// 40 Visualizations/CLIENT/SERIAL Client/SERIAL Client/POPUP/PARAMETER/VIS_ModBusParameter_SERIAL_Client
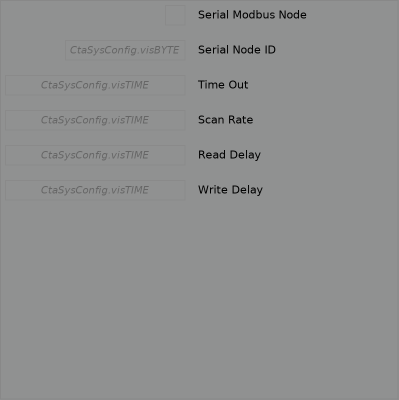
VISUALIZATION VIS_ModBusParameter_SERIAL_Client  // 399x400
VAR_IN_OUT
    fbMbSerialClientIn   : fbMbSerialClient; 
END_VAR
    Label (195,5 195x20), "Serial Modbus Node"
    Label (195,40 195x20), "Serial Node ID"
    Frame (65,40 120x20)
        shows CtaSysConfig.visBYTE(visfbBYTEIn := fbMbSerialClientIn.scParameter.fbbyUnitId)
    Frame (165,5 20x20)
        shows CtaSysConfig.visBOOL(visfbBOOLIn := fbMbSerialClientIn.scParameter.fbxEnable)
    Label (195,75 195x20), "Time Out"
    Frame (5,75 180x20)
        shows CtaSysConfig.visTIME(visfbTIMEIn := fbMbSerialClientIn.scParameter.fbtTimeOut)
    Frame (5,110 180x20)
        shows CtaSysConfig.visTIME(visfbTIMEIn := fbMbSerialClientIn.scParameter.fbtScanRate)
    Label (195,110 195x20), "Scan Rate"
    Frame (5,145 180x20)
        shows CtaSysConfig.visTIME(visfbTIMEIn := fbMbSerialClientIn.scParameter.fbtDelayRead)
    Label (195,145 195x20), "Read Delay"
    Frame (5,180 180x20)
        shows CtaSysConfig.visTIME(visfbTIMEIn := fbMbSerialClientIn.scParameter.fbtDelayWrite)
    Label (195,180 195x20), "Write Delay"
END_VISUALIZATION

// 40 Visualizations/CLIENT/NETWORK Client/TCP/VIS_ModBusTcpNode_QUERRY
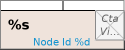
VISUALIZATION VIS_ModBusTcpNode_QUERRY  // 125x50
VAR_IN_OUT
	fbMbTcpClientIn   : REFERENCE TO fbMbTcpClient;      
END_VAR
    RoundedRectangle (0,10 125x40), colour toggle: fbMbTcpClientIn.xError
    RoundedRectangle (0,10 125x40), colour toggle: fbMbTcpClientIn.xError, invisible if: fbMbTcpClientIn.xComAktive
    Image (95,10 30x30), image: CtaVisSymbols.ImagePool.gear
        OnMouseClick:  Dialog=VIS_ModBus_Tcpl_NodePopUp, Parameters={fbMbTcpClientIn: fbMbTcpClientIn}, Selected={0: }, OpenModal=True, OpenCentered=True
    Textfield (30,37 90x10), "Node Id %d", text variable: fbMbTcpClientIn.byUnitId, invisible if: NOT __ISVALIDREF(fbMbTcpClientIn)
    Line (63,10) (63,0)
    Frame (5,15 80x20)
        shows Node_BMK(ITF_BMK := fbMbTcpClientIn.proITF_BMK)
END_VISUALIZATION

// 40 Visualizations/CLIENT/NETWORK Client/TCP/VIS_ModBusTcpNode
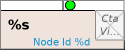
VISUALIZATION VIS_ModBusTcpNode  // 125x50
VAR_INPUT   
	ITF_TCP_NODEIN :   ITF_TCP_NODE;   
    xCourrentNode     :   BOOL;
END_VAR
    Frame (0,0 125x50), invisible if: NOT __QUERYINTERFACE(ITF_TCP_NODEIN,ITF_TCP_NODEIN)
        shows VIS_ModBusTcpNode_QUERRY(fbMbTcpClientIn := ITF_TCP_NODEIN.proNodeReference)
    Ellipse (65,0 10x10), invisible if: NOT xCourrentNode
END_VISUALIZATION

// 40 Visualizations/CLIENT/NETWORK Client/TCP/POPUP/VIS_ModBus_Tcpl_NodePopUp
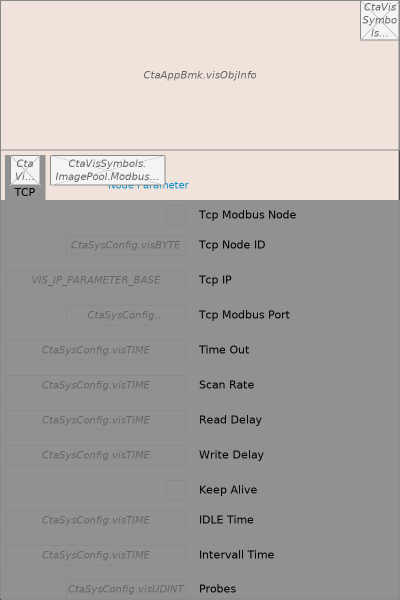
VISUALIZATION VIS_ModBus_Tcpl_NodePopUp  // 400x600
VAR_IN_OUT
    {attribute 'VAR_IN_OUT_AS_POINTER'}
	fbMbTcpClientIn   : fbMbTcpClient; 
END_VAR
    Rectangle (0,0 400x600)
    Label (105,180 150x10), "Node Parameter"
    Image (50,155 115x30), image: CtaVisSymbols.ImagePool.Modbus_Organization_Logo
    Group (5,155 40x45)
        Rectangle (0,0 40x45)
        Label (5,30 30x15), "TCP"
        Image (5,0 30x30), image: CtaVisSymbols.ImagePool.lan
    Frame (1,200 399x400)
        shows VIS_ModBusParameter_TCP_Client(fbMbTcpClientIn := fbMbTcpClientIn)
        shows VIS_ModBusParameter_UDP(fbModBusServerIn := fbModBusServerIn)
        shows VIS_ModBusParameter_SERIAL(fbModBusServerIn := fbModBusServerIn)
    Image (360,0 40x40), image: CtaVisSymbols.ImagePool.close_solo_black
        OnMouseClick:  Dialog=VIS_ModBus_Tcpl_NodePopUp, Result=None, NumpadKeypadSet=True
    Frame (0,0 400x150)
        shows CtaAppBmk.visObjInfo(ITF_BMK_IN := fbMbTcpClientIn.proITF_BMK)
END_VISUALIZATION

// 40 Visualizations/CLIENT/NETWORK Client/TCP/POPUP/PARAMETER/VIS_ModBusParameter_TCP_Client
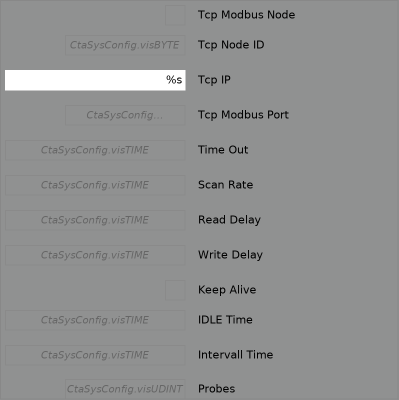
VISUALIZATION VIS_ModBusParameter_TCP_Client  // 399x400
VAR_IN_OUT
    fbMbTcpClientIn   : fbMbTcpClient; 
END_VAR
    Label (195,5 195x20), "Tcp Modbus Node"
    Label (195,35 195x20), "Tcp Node ID"
    Frame (65,35 120x20)
        shows CtaSysConfig.visBYTE(visfbBYTEIn := fbMbTcpClientIn.scParameter.fbbyUnitId)
    Frame (165,5 20x20)
        shows CtaSysConfig.visBOOL(visfbBOOLIn := fbMbTcpClientIn.scParameter.fbxEnable)
    Label (195,140 195x20), "Time Out"
    Frame (5,140 180x20)
        shows CtaSysConfig.visTIME(visfbTIMEIn := fbMbTcpClientIn.scParameter.fbtTimeOut)
    Frame (5,175 180x20)
        shows CtaSysConfig.visTIME(visfbTIMEIn := fbMbTcpClientIn.scParameter.fbtScanRate)
    Label (195,175 195x20), "Scan Rate"
    Frame (5,70 180x20)
        shows VIS_IP_PARAMETER(ITF_STRING40In := fbMbTcpClientIn.scParameter.fbstIp)
    Label (195,70 195x20), "Tcp IP"
    Frame (65,105 120x20)
        shows CtaSysConfig.visWORD_DEZ(visfbWORDIn := fbMbTcpClientIn.scParameter.fbwPort)
    Label (195,105 195x20), "Tcp Modbus Port"
    Frame (165,280 20x20)
        shows CtaSysConfig.visBOOL(visfbBOOLIn := fbMbTcpClientIn.scParameter.fbxKeepAlive)
    Label (195,280 195x20), "Keep Alive"
    Frame (5,310 180x20)
        shows CtaSysConfig.visTIME(visfbTIMEIn := fbMbTcpClientIn.scParameter.fbtMaxIdleTime)
    Label (195,310 195x20), "IDLE Time"
    Label (195,345 195x20), "Intervall Time"
    Frame (5,345 180x20)
        shows CtaSysConfig.visTIME(visfbTIMEIn := fbMbTcpClientIn.scParameter.fbtIntervall)
    Frame (65,379 120x20)
        shows CtaSysConfig.visUDINT(visfbUDINTIn := fbMbTcpClientIn.scParameter.fbudiProbes)
    Label (195,379 195x20), "Probes"
    Frame (5,210 180x20)
        shows CtaSysConfig.visTIME(visfbTIMEIn := fbMbTcpClientIn.scParameter.fbtDelayRead)
    Label (195,210 195x20), "Read Delay"
    Frame (5,245 180x20)
        shows CtaSysConfig.visTIME(visfbTIMEIn := fbMbTcpClientIn.scParameter.fbtDelayWrite)
    Label (195,245 195x20), "Write Delay"
END_VISUALIZATION

// 40 Visualizations/CLIENT/NETWORK Client/VIS_MODBUS_TCP_LINE
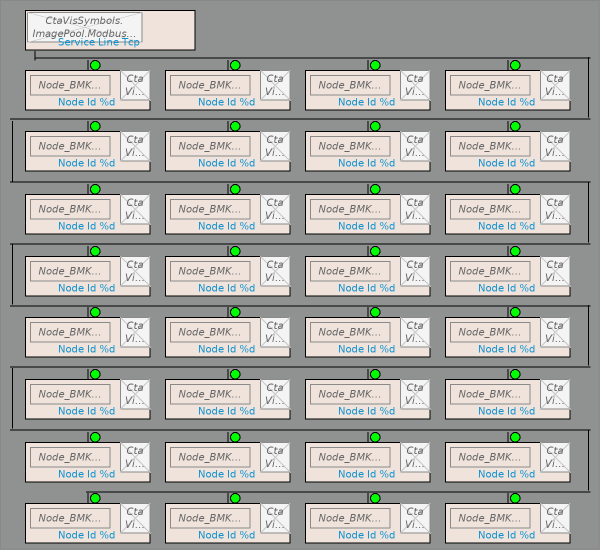
VISUALIZATION VIS_MODBUS_TCP_LINE  // 600x550
VAR_IN_OUT
	fbMbTcpPortControll   : fbMbTcpPortControll;      
END_VAR
    Frame (509,56 81x4), invisible if: fbMbTcpPortControll.bCountetCalls < 5
        shows VIS_TCP_LINE_HORIZONTAL()
    Frame (369,56 141x4), invisible if: fbMbTcpPortControll.bCountetCalls < 4
        shows VIS_TCP_LINE_HORIZONTAL()
    Frame (25,10 170x50)
        shows VIS_ModBusNetworkPortTcp(fbMbTcpPortControllIn := fbMbTcpPortControll)
    Frame (194,56 36x4), invisible if: fbMbTcpPortControll.bCountetCalls < 2
        shows VIS_TCP_LINE_HORIZONTAL()
    Frame (586,57 4x60), invisible if: fbMbTcpPortControll.bCountetCalls < 5
        shows VIS_TCP_LINE_VERTIKAL()
    Frame (10,121 4x60), invisible if: fbMbTcpPortControll.bCountetCalls < 9
        shows VIS_TCP_LINE_VERTIKAL()
    Frame (10,180 80x4), invisible if: fbMbTcpPortControll.bCountetCalls < 9
        shows VIS_TCP_LINE_HORIZONTAL()
    Frame (586,182 4x60), invisible if: fbMbTcpPortControll.bCountetCalls < 13
        shows VIS_TCP_LINE_VERTIKAL()
    Frame (10,244 4x60), invisible if: fbMbTcpPortControll.bCountetCalls < 17
        shows VIS_TCP_LINE_VERTIKAL()
    Frame (586,305 4x60), invisible if: fbMbTcpPortControll.bCountetCalls < 21
        shows VIS_TCP_LINE_VERTIKAL()
    Frame (10,368 4x60), invisible if: fbMbTcpPortControll.bCountetCalls < 25
        shows VIS_TCP_LINE_VERTIKAL()
    Frame (586,430 4x60), invisible if: fbMbTcpPortControll.bCountetCalls < 29
        shows VIS_TCP_LINE_VERTIKAL()
    Frame (229,56 141x4), invisible if: fbMbTcpPortControll.bCountetCalls < 3
        shows VIS_TCP_LINE_HORIZONTAL()
    Frame (506,117 84x4), invisible if: fbMbTcpPortControll.bCountetCalls < 5
        shows VIS_TCP_LINE_HORIZONTAL()
    Frame (366,117 141x4), invisible if: fbMbTcpPortControll.bCountetCalls < 6
        shows VIS_TCP_LINE_HORIZONTAL()
    Frame (86,117 141x4), invisible if: fbMbTcpPortControll.bCountetCalls < 8
        shows VIS_TCP_LINE_HORIZONTAL()
    Frame (226,117 141x4), invisible if: fbMbTcpPortControll.bCountetCalls < 7
        shows VIS_TCP_LINE_HORIZONTAL()
    Frame (10,117 77x4), invisible if: fbMbTcpPortControll.bCountetCalls < 9
        shows VIS_TCP_LINE_HORIZONTAL()
    Frame (89,180 141x4), invisible if: fbMbTcpPortControll.bCountetCalls < 10
        shows VIS_TCP_LINE_HORIZONTAL()
    Frame (229,180 141x4), invisible if: fbMbTcpPortControll.bCountetCalls < 11
        shows VIS_TCP_LINE_HORIZONTAL()
    Frame (509,180 81x4), invisible if: fbMbTcpPortControll.bCountetCalls < 13
        shows VIS_TCP_LINE_HORIZONTAL()
    Frame (369,180 141x4), invisible if: fbMbTcpPortControll.bCountetCalls < 12
        shows VIS_TCP_LINE_HORIZONTAL()
    Frame (506,242 84x4), invisible if: fbMbTcpPortControll.bCountetCalls < 13
        shows VIS_TCP_LINE_HORIZONTAL()
    Frame (366,242 141x4), invisible if: fbMbTcpPortControll.bCountetCalls < 14
        shows VIS_TCP_LINE_HORIZONTAL()
    Frame (86,242 141x4), invisible if: fbMbTcpPortControll.bCountetCalls < 16
        shows VIS_TCP_LINE_HORIZONTAL()
    Frame (226,242 141x4), invisible if: fbMbTcpPortControll.bCountetCalls < 15
        shows VIS_TCP_LINE_HORIZONTAL()
    Frame (10,242 77x4), invisible if: fbMbTcpPortControll.bCountetCalls < 17
        shows VIS_TCP_LINE_HORIZONTAL()
    Frame (10,304 80x4), invisible if: fbMbTcpPortControll.bCountetCalls < 17
        shows VIS_TCP_LINE_HORIZONTAL()
    Frame (89,304 141x4), invisible if: fbMbTcpPortControll.bCountetCalls < 18
        shows VIS_TCP_LINE_HORIZONTAL()
    Frame (229,304 141x4), invisible if: fbMbTcpPortControll.bCountetCalls < 19
        shows VIS_TCP_LINE_HORIZONTAL()
    Frame (509,304 81x4), invisible if: fbMbTcpPortControll.bCountetCalls < 21
        shows VIS_TCP_LINE_HORIZONTAL()
    Frame (369,304 141x4), invisible if: fbMbTcpPortControll.bCountetCalls < 20
        shows VIS_TCP_LINE_HORIZONTAL()
    Frame (506,365 84x4), invisible if: fbMbTcpPortControll.bCountetCalls < 21
        shows VIS_TCP_LINE_HORIZONTAL()
    Frame (366,365 141x4), invisible if: fbMbTcpPortControll.bCountetCalls < 22
        shows VIS_TCP_LINE_HORIZONTAL()
    Frame (86,365 141x4), invisible if: fbMbTcpPortControll.bCountetCalls < 24
        shows VIS_TCP_LINE_HORIZONTAL()
    Frame (226,365 141x4), invisible if: fbMbTcpPortControll.bCountetCalls < 23
        shows VIS_TCP_LINE_HORIZONTAL()
    Frame (10,365 77x4), invisible if: fbMbTcpPortControll.bCountetCalls < 25
        shows VIS_TCP_LINE_HORIZONTAL()
    Frame (10,428 80x4), invisible if: fbMbTcpPortControll.bCountetCalls < 25
        shows VIS_TCP_LINE_HORIZONTAL()
    Frame (89,428 141x4), invisible if: fbMbTcpPortControll.bCountetCalls < 26
        shows VIS_TCP_LINE_HORIZONTAL()
    Frame (229,428 141x4), invisible if: fbMbTcpPortControll.bCountetCalls < 27
        shows VIS_TCP_LINE_HORIZONTAL()
    Frame (509,428 81x4), invisible if: fbMbTcpPortControll.bCountetCalls < 29
        shows VIS_TCP_LINE_HORIZONTAL()
    Frame (369,428 141x4), invisible if: fbMbTcpPortControll.bCountetCalls < 28
        shows VIS_TCP_LINE_HORIZONTAL()
    Frame (506,490 84x4), invisible if: fbMbTcpPortControll.bCountetCalls < 29
        shows VIS_TCP_LINE_HORIZONTAL()
    Frame (366,490 141x4), invisible if: fbMbTcpPortControll.bCountetCalls < 30
        shows VIS_TCP_LINE_HORIZONTAL()
    Frame (86,490 141x4), invisible if: fbMbTcpPortControll.bCountetCalls < 32
        shows VIS_TCP_LINE_HORIZONTAL()
    Frame (226,490 141x4), invisible if: fbMbTcpPortControll.bCountetCalls < 31
        shows VIS_TCP_LINE_HORIZONTAL()
    Frame (25,60 125x50), invisible if: NOT fbMbTcpPortControll.ayShowNodes[1]
        shows VIS_ModBusTcpNode(ITF_TCP_NODEIN := fbMbTcpPortControll.ayNodes[1], xCourrentNode := fbMbTcpPortControll.bIdOfCourrentCall = 1)
        shows VIS_ModBusTcpNode()
        p1371288417: fbMbSerialPortControllIn.ayNodes[1]
    Frame (305,60 125x50), invisible if: NOT fbMbTcpPortControll.ayShowNodes[3]
        shows VIS_ModBusTcpNode(ITF_TCP_NODEIN := fbMbTcpPortControll.ayNodes[3], xCourrentNode := fbMbTcpPortControll.bIdOfCourrentCall = 3)
        shows VIS_ModBusTcpNode(ITF_TCP_NODEIN := fbMbTcpPortControll.ayNodes[3], xCourrentNode := fbMbTcpPortControll.bIdOfCourrentCall = 3)
        p1371288417: fbMbTcpPortControll.ayNodes[3]
    Frame (445,60 125x50), invisible if: NOT fbMbTcpPortControll.ayShowNodes[4]
        shows VIS_ModBusTcpNode(ITF_TCP_NODEIN := fbMbTcpPortControll.ayNodes[4], xCourrentNode := fbMbTcpPortControll.bIdOfCourrentCall = 4)
        shows VIS_ModBusTcpNode(ITF_TCP_NODEIN := fbMbTcpPortControll.ayNodes[4], xCourrentNode := fbMbTcpPortControll.bIdOfCourrentCall = 4)
        p1371288417: fbMbTcpPortControll.ayNodes[4]
    Frame (445,184 125x50), invisible if: NOT fbMbTcpPortControll.ayShowNodes[12]
        shows VIS_ModBusTcpNode(ITF_TCP_NODEIN := fbMbTcpPortControll.ayNodes[12], xCourrentNode := fbMbTcpPortControll.bIdOfCourrentCall = 12)
        shows VIS_ModBusTcpNode(ITF_TCP_NODEIN := fbMbTcpPortControll.ayNodes[12], xCourrentNode := fbMbTcpPortControll.bIdOfCourrentCall = 12)
        p1371288417: fbMbTcpPortControll.ayNodes[12]
    Frame (25,184 125x50), invisible if: NOT fbMbTcpPortControll.ayShowNodes[9]
        shows VIS_ModBusTcpNode(ITF_TCP_NODEIN := fbMbTcpPortControll.ayNodes[9], xCourrentNode := fbMbTcpPortControll.bIdOfCourrentCall = 9)
        shows VIS_ModBusTcpNode(ITF_TCP_NODEIN := fbMbTcpPortControll.ayNodes[9], xCourrentNode := fbMbTcpPortControll.bIdOfCourrentCall = 9)
        p1371288417: fbMbTcpPortControll.ayNodes[9]
    Frame (165,184 125x50), invisible if: NOT fbMbTcpPortControll.ayShowNodes[10]
        shows VIS_ModBusTcpNode(ITF_TCP_NODEIN := fbMbTcpPortControll.ayNodes[10], xCourrentNode := fbMbTcpPortControll.bIdOfCourrentCall = 10)
        shows VIS_ModBusTcpNode(ITF_TCP_NODEIN := fbMbTcpPortControll.ayNodes[10], xCourrentNode := fbMbTcpPortControll.bIdOfCourrentCall = 10)
        p1371288417: fbMbTcpPortControll.ayNodes[10]
    Frame (305,184 125x50), invisible if: NOT fbMbTcpPortControll.ayShowNodes[11]
        shows VIS_ModBusTcpNode(ITF_TCP_NODEIN := fbMbTcpPortControll.ayNodes[11], xCourrentNode := fbMbTcpPortControll.bIdOfCourrentCall = 11)
        shows VIS_ModBusTcpNode(ITF_TCP_NODEIN := fbMbTcpPortControll.ayNodes[11], xCourrentNode := fbMbTcpPortControll.bIdOfCourrentCall = 11)
        p1371288417: fbMbTcpPortControll.ayNodes[11]
    Frame (25,369 125x50), invisible if: NOT fbMbTcpPortControll.ayShowNodes[24]
        shows VIS_ModBusTcpNode(ITF_TCP_NODEIN := fbMbTcpPortControll.ayNodes[24], xCourrentNode := fbMbTcpPortControll.bIdOfCourrentCall = 24)
        shows VIS_ModBusTcpNode(ITF_TCP_NODEIN := fbMbTcpPortControll.ayNodes[24], xCourrentNode := fbMbTcpPortControll.bIdOfCourrentCall = 24)
        p1371288417: fbMbTcpPortControll.ayNodes[24]
    Frame (165,369 125x50), invisible if: NOT fbMbTcpPortControll.ayShowNodes[23]
        shows VIS_ModBusTcpNode(ITF_TCP_NODEIN := fbMbTcpPortControll.ayNodes[23], xCourrentNode := fbMbTcpPortControll.bIdOfCourrentCall = 23)
        shows VIS_ModBusTcpNode(ITF_TCP_NODEIN := fbMbTcpPortControll.ayNodes[23], xCourrentNode := fbMbTcpPortControll.bIdOfCourrentCall = 23)
        p1371288417: fbMbTcpPortControll.ayNodes[23]
    Frame (305,369 125x50), invisible if: NOT fbMbTcpPortControll.ayShowNodes[22]
        shows VIS_ModBusTcpNode(ITF_TCP_NODEIN := fbMbTcpPortControll.ayNodes[22], xCourrentNode := fbMbTcpPortControll.bIdOfCourrentCall = 22)
        shows VIS_ModBusTcpNode(ITF_TCP_NODEIN := fbMbTcpPortControll.ayNodes[22], xCourrentNode := fbMbTcpPortControll.bIdOfCourrentCall = 22)
        p1371288417: fbMbTcpPortControll.ayNodes[22]
    Frame (445,369 125x50), invisible if: NOT fbMbTcpPortControll.ayShowNodes[21]
        shows VIS_ModBusTcpNode(ITF_TCP_NODEIN := fbMbTcpPortControll.ayNodes[21], xCourrentNode := fbMbTcpPortControll.bIdOfCourrentCall = 21)
        shows VIS_ModBusTcpNode(ITF_TCP_NODEIN := fbMbTcpPortControll.ayNodes[21], xCourrentNode := fbMbTcpPortControll.bIdOfCourrentCall = 21)
        p1371288417: fbMbTcpPortControll.ayNodes[21]
    Frame (445,432 125x50), invisible if: NOT fbMbTcpPortControll.ayShowNodes[28]
        shows VIS_ModBusTcpNode(ITF_TCP_NODEIN := fbMbTcpPortControll.ayNodes[28], xCourrentNode := fbMbTcpPortControll.bIdOfCourrentCall = 28)
        shows VIS_ModBusTcpNode(ITF_TCP_NODEIN := fbMbTcpPortControll.ayNodes[28], xCourrentNode := fbMbTcpPortControll.bIdOfCourrentCall = 28)
        p1371288417: fbMbTcpPortControll.ayNodes[28]
    Frame (25,432 125x50), invisible if: NOT fbMbTcpPortControll.ayShowNodes[25]
        shows VIS_ModBusTcpNode(ITF_TCP_NODEIN := fbMbTcpPortControll.ayNodes[25], xCourrentNode := fbMbTcpPortControll.bIdOfCourrentCall = 25)
        shows VIS_ModBusTcpNode(ITF_TCP_NODEIN := fbMbTcpPortControll.ayNodes[25], xCourrentNode := fbMbTcpPortControll.bIdOfCourrentCall = 25)
        p1371288417: fbMbTcpPortControll.ayNodes[25]
    Frame (165,432 125x50), invisible if: NOT fbMbTcpPortControll.ayShowNodes[26]
        shows VIS_ModBusTcpNode(ITF_TCP_NODEIN := fbMbTcpPortControll.ayNodes[26], xCourrentNode := fbMbTcpPortControll.bIdOfCourrentCall = 26)
        shows VIS_ModBusTcpNode(ITF_TCP_NODEIN := fbMbTcpPortControll.ayNodes[26], xCourrentNode := fbMbTcpPortControll.bIdOfCourrentCall = 26)
        p1371288417: fbMbTcpPortControll.ayNodes[26]
    Frame (305,432 125x50), invisible if: NOT fbMbTcpPortControll.ayShowNodes[27]
        shows VIS_ModBusTcpNode(ITF_TCP_NODEIN := fbMbTcpPortControll.ayNodes[27], xCourrentNode := fbMbTcpPortControll.bIdOfCourrentCall = 27)
        shows VIS_ModBusTcpNode(ITF_TCP_NODEIN := fbMbTcpPortControll.ayNodes[27], xCourrentNode := fbMbTcpPortControll.bIdOfCourrentCall = 27)
        p1371288417: fbMbTcpPortControll.ayNodes[27]
    Frame (25,493 125x50), invisible if: NOT fbMbTcpPortControll.ayShowNodes[32]
        shows VIS_ModBusTcpNode(ITF_TCP_NODEIN := fbMbTcpPortControll.ayNodes[32], xCourrentNode := fbMbTcpPortControll.bIdOfCourrentCall = 32)
        shows VIS_ModBusTcpNode(ITF_TCP_NODEIN := fbMbTcpPortControll.ayNodes[32], xCourrentNode := fbMbTcpPortControll.bIdOfCourrentCall = 32)
        p1371288417: fbMbTcpPortControll.ayNodes[32]
    Frame (165,493 125x50), invisible if: NOT fbMbTcpPortControll.ayShowNodes[31]
        shows VIS_ModBusTcpNode(ITF_TCP_NODEIN := fbMbTcpPortControll.ayNodes[31], xCourrentNode := fbMbTcpPortControll.bIdOfCourrentCall = 31)
        shows VIS_ModBusTcpNode(ITF_TCP_NODEIN := fbMbTcpPortControll.ayNodes[31], xCourrentNode := fbMbTcpPortControll.bIdOfCourrentCall = 31)
        p1371288417: fbMbTcpPortControll.ayNodes[31]
    Frame (305,493 125x50), invisible if: NOT fbMbTcpPortControll.ayShowNodes[30]
        shows VIS_ModBusTcpNode(ITF_TCP_NODEIN := fbMbTcpPortControll.ayNodes[30], xCourrentNode := fbMbTcpPortControll.bIdOfCourrentCall = 30)
        shows VIS_ModBusTcpNode(ITF_TCP_NODEIN := fbMbTcpPortControll.ayNodes[30], xCourrentNode := fbMbTcpPortControll.bIdOfCourrentCall = 30)
        p1371288417: fbMbTcpPortControll.ayNodes[30]
    Frame (445,493 125x50), invisible if: NOT fbMbTcpPortControll.ayShowNodes[29]
        shows VIS_ModBusTcpNode(ITF_TCP_NODEIN := fbMbTcpPortControll.ayNodes[29], xCourrentNode := fbMbTcpPortControll.bIdOfCourrentCall = 29)
        shows VIS_ModBusTcpNode(ITF_TCP_NODEIN := fbMbTcpPortControll.ayNodes[29], xCourrentNode := fbMbTcpPortControll.bIdOfCourrentCall = 29)
        p1371288417: fbMbTcpPortControll.ayNodes[29]
    Frame (165,60 125x50), invisible if: NOT fbMbTcpPortControll.ayShowNodes[2]
        shows VIS_ModBusTcpNode(ITF_TCP_NODEIN := fbMbTcpPortControll.ayNodes[2], xCourrentNode := fbMbTcpPortControll.bIdOfCourrentCall = 2)
        shows VIS_ModBusTcpNode(ITF_TCP_NODEIN := fbMbTcpPortControll.ayNodes[2], xCourrentNode := fbMbTcpPortControll.bIdOfCourrentCall = 2)
        p1371288417: fbMbTcpPortControll.ayNodes[2]
    Frame (445,121 125x50), invisible if: NOT fbMbTcpPortControll.ayShowNodes[5]
        shows VIS_ModBusTcpNode(ITF_TCP_NODEIN := fbMbTcpPortControll.ayNodes[5], xCourrentNode := fbMbTcpPortControll.bIdOfCourrentCall = 5)
        shows VIS_ModBusTcpNode(ITF_TCP_NODEIN := fbMbTcpPortControll.ayNodes[5], xCourrentNode := fbMbTcpPortControll.bIdOfCourrentCall = 5)
        p1371288417: fbMbTcpPortControll.ayNodes[5]
    Frame (165,121 125x50), invisible if: NOT fbMbTcpPortControll.ayShowNodes[7]
        shows VIS_ModBusTcpNode(ITF_TCP_NODEIN := fbMbTcpPortControll.ayNodes[7], xCourrentNode := fbMbTcpPortControll.bIdOfCourrentCall = 7)
        shows VIS_ModBusTcpNode(ITF_TCP_NODEIN := fbMbTcpPortControll.ayNodes[7], xCourrentNode := fbMbTcpPortControll.bIdOfCourrentCall = 7)
        p1371288417: fbMbTcpPortControll.ayNodes[7]
    Frame (25,121 125x50), invisible if: NOT fbMbTcpPortControll.ayShowNodes[8]
        shows VIS_ModBusTcpNode(ITF_TCP_NODEIN := fbMbTcpPortControll.ayNodes[8], xCourrentNode := fbMbTcpPortControll.bIdOfCourrentCall = 8)
        shows VIS_ModBusTcpNode(ITF_TCP_NODEIN := fbMbTcpPortControll.ayNodes[8], xCourrentNode := fbMbTcpPortControll.bIdOfCourrentCall = 8)
        p1371288417: fbMbTcpPortControll.ayNodes[8]
    Frame (305,121 125x50), invisible if: NOT fbMbTcpPortControll.ayShowNodes[6]
        shows VIS_ModBusTcpNode(ITF_TCP_NODEIN := fbMbTcpPortControll.ayNodes[6], xCourrentNode := fbMbTcpPortControll.bIdOfCourrentCall = 6)
        shows VIS_ModBusTcpNode(ITF_TCP_NODEIN := fbMbTcpPortControll.ayNodes[6], xCourrentNode := fbMbTcpPortControll.bIdOfCourrentCall = 6)
        p1371288417: fbMbTcpPortControll.ayNodes[6]
    Frame (445,246 125x50), invisible if: NOT fbMbTcpPortControll.ayShowNodes[13]
        shows VIS_ModBusTcpNode(ITF_TCP_NODEIN := fbMbTcpPortControll.ayNodes[13], xCourrentNode := fbMbTcpPortControll.bIdOfCourrentCall = 13)
        shows VIS_ModBusTcpNode(ITF_TCP_NODEIN := fbMbTcpPortControll.ayNodes[13], xCourrentNode := fbMbTcpPortControll.bIdOfCourrentCall = 13)
        p1371288417: fbMbTcpPortControll.ayNodes[13]
    Frame (305,246 125x50), invisible if: NOT fbMbTcpPortControll.ayShowNodes[14]
        shows VIS_ModBusTcpNode(ITF_TCP_NODEIN := fbMbTcpPortControll.ayNodes[14], xCourrentNode := fbMbTcpPortControll.bIdOfCourrentCall = 14)
        shows VIS_ModBusTcpNode(ITF_TCP_NODEIN := fbMbTcpPortControll.ayNodes[14], xCourrentNode := fbMbTcpPortControll.bIdOfCourrentCall = 14)
        p1371288417: fbMbTcpPortControll.ayNodes[14]
    Frame (165,246 125x50), invisible if: NOT fbMbTcpPortControll.ayShowNodes[15]
        shows VIS_ModBusTcpNode(ITF_TCP_NODEIN := fbMbTcpPortControll.ayNodes[15], xCourrentNode := fbMbTcpPortControll.bIdOfCourrentCall = 15)
        shows VIS_ModBusTcpNode(ITF_TCP_NODEIN := fbMbTcpPortControll.ayNodes[15], xCourrentNode := fbMbTcpPortControll.bIdOfCourrentCall = 15)
        p1371288417: fbMbTcpPortControll.ayNodes[15]
    Frame (25,246 125x50), invisible if: NOT fbMbTcpPortControll.ayShowNodes[16]
        shows VIS_ModBusTcpNode(ITF_TCP_NODEIN := fbMbTcpPortControll.ayNodes[16], xCourrentNode := fbMbTcpPortControll.bIdOfCourrentCall = 16)
        shows VIS_ModBusTcpNode(ITF_TCP_NODEIN := fbMbTcpPortControll.ayNodes[16], xCourrentNode := fbMbTcpPortControll.bIdOfCourrentCall = 16)
        p1371288417: fbMbTcpPortControll.ayNodes[16]
    Frame (25,307 125x50), invisible if: NOT fbMbTcpPortControll.ayShowNodes[17]
        shows VIS_ModBusTcpNode(ITF_TCP_NODEIN := fbMbTcpPortControll.ayNodes[17], xCourrentNode := fbMbTcpPortControll.bIdOfCourrentCall = 17)
        shows VIS_ModBusTcpNode(ITF_TCP_NODEIN := fbMbTcpPortControll.ayNodes[17], xCourrentNode := fbMbTcpPortControll.bIdOfCourrentCall = 17)
        p1371288417: fbMbTcpPortControll.ayNodes[17]
    Frame (445,307 125x50), invisible if: NOT fbMbTcpPortControll.ayShowNodes[20]
        shows VIS_ModBusTcpNode(ITF_TCP_NODEIN := fbMbTcpPortControll.ayNodes[20], xCourrentNode := fbMbTcpPortControll.bIdOfCourrentCall = 20)
        shows VIS_ModBusTcpNode(ITF_TCP_NODEIN := fbMbTcpPortControll.ayNodes[20], xCourrentNode := fbMbTcpPortControll.bIdOfCourrentCall = 20)
        p1371288417: fbMbTcpPortControll.ayNodes[20]
    Frame (165,307 125x50), invisible if: NOT fbMbTcpPortControll.ayShowNodes[18]
        shows VIS_ModBusTcpNode(ITF_TCP_NODEIN := fbMbTcpPortControll.ayNodes[18], xCourrentNode := fbMbTcpPortControll.bIdOfCourrentCall = 18)
        shows VIS_ModBusTcpNode(ITF_TCP_NODEIN := fbMbTcpPortControll.ayNodes[18], xCourrentNode := fbMbTcpPortControll.bIdOfCourrentCall = 18)
        p1371288417: fbMbTcpPortControll.ayNodes[18]
    Frame (305,307 125x50), invisible if: NOT fbMbTcpPortControll.ayShowNodes[19]
        shows VIS_ModBusTcpNode(ITF_TCP_NODEIN := fbMbTcpPortControll.ayNodes[19], xCourrentNode := fbMbTcpPortControll.bIdOfCourrentCall = 19)
        shows VIS_ModBusTcpNode(ITF_TCP_NODEIN := fbMbTcpPortControll.ayNodes[19], xCourrentNode := fbMbTcpPortControll.bIdOfCourrentCall = 19)
        p1371288417: fbMbTcpPortControll.ayNodes[19]
END_VISUALIZATION

// 40 Visualizations/CLIENT/NETWORK Client/VIS_TCP_LINE_HORIZONTAL
VISUALIZATION VIS_TCP_LINE_HORIZONTAL  // 100x4
    Line (100,2) (0,2)
END_VISUALIZATION

// 40 Visualizations/CLIENT/NETWORK Client/VIS_TCP_LINE_VERTIKAL
VISUALIZATION VIS_TCP_LINE_VERTIKAL  // 4x100
    Line (2,0) (2,100)
END_VISUALIZATION

// 40 Visualizations/CLIENT/VIS_MODBUS_LINE
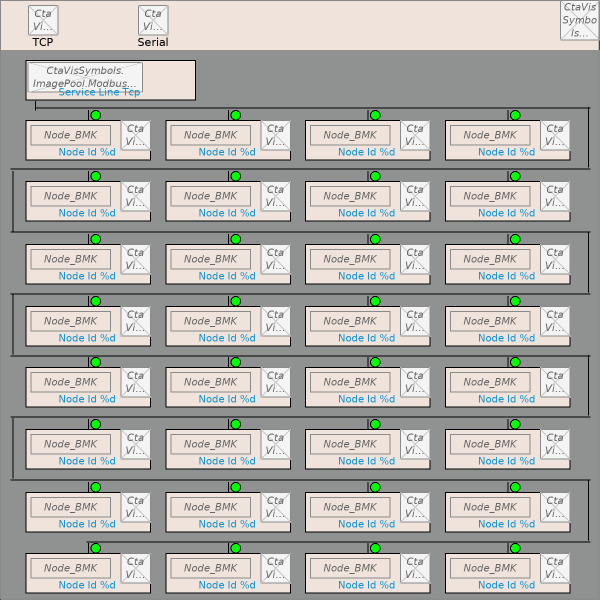
VISUALIZATION VIS_MODBUS_LINE  // 600x600
VAR_IN_OUT
	{attribute 'VAR_IN_OUT_AS_POINTER'}
	fbMbTcpPortControllIn   	: fbMbTcpPortControll;
	{attribute 'VAR_IN_OUT_AS_POINTER'}  
    fbMbSerialPortControllIn   	: fbMbSerialPortControll;         
END_VAR
VAR
    usiTcpSerial        :   USINT;
END_VAR
    Rectangle (0,0 600x600)
    Frame (1,50 599x550), frame switch variable: usiTcpSerial
        shows VIS_MODBUS_TCP_LINE(fbMbTcpPortControll := fbMbTcpPortControllIn)
        shows VIS_MODBUS_SERIAL_LINE(fbMbSerialPortControllIn := fbMbSerialPortControllIn)
    Group (23,5 40x45)
        OnMouseClick: execute { usiTcpSerial := 0; }
        Rectangle (0,0 40x45), colour toggle: usiTcpSerial = 0
        Image (5,0 30x30), image: CtaVisSymbols.ImagePool.lan
        Label (5,30 30x15), "TCP"
    Group (133,5 40x45)
        OnMouseClick: execute { usiTcpSerial := 1; }
        Rectangle (0,0 40x45), colour toggle: usiTcpSerial = 1
        Image (5,0 30x30), image: CtaVisSymbols.ImagePool.lan
        Label (5,30 30x15), "Serial"
    Image (560,0 40x40), image: CtaVisSymbols.ImagePool.close_solo_black
        OnMouseClick:  Dialog=Current Dialog, Result=OK, NumpadKeypadSet=True
END_VISUALIZATION

// 40 Visualizations/BMK/Node_BMK
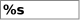
VISUALIZATION Node_BMK  // 80x20
VAR_INPUT
	ITF_BMK : CtaAppBmk.ITF_BMK;
END_VAR
    Frame (0,0 80x20), invisible if: NOT __QUERYINTERFACE(ITF_BMK,ITF_BMK)
        shows Node_BMK_QUERY(ITF_BMK := ITF_BMK)
END_VISUALIZATION

// 40 Visualizations/BMK/Node_BMK_QUERY
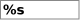
VISUALIZATION Node_BMK_QUERY  // 80x20
VAR_INPUT
	ITF_BMK : CtaAppBmk.ITF_BMK;
END_VAR
    Textfield (0,0 80x20), "%s", text variable: ITF_BMK.proGetBMK, invisible if: NOT __QUERYINTERFACE(ITF_BMK,ITF_BMK)
END_VISUALIZATION

// 40 Visualizations/DIALOG/ModBusPopUp
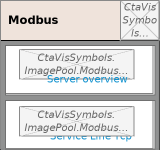
VISUALIZATION ModBusPopUp  // 160x150
VAR_IN_OUT
	{attribute 'VAR_IN_OUT_AS_POINTER'}
	fbModBusServerIn   			:	fbModBusServer; 
	{attribute 'VAR_IN_OUT_AS_POINTER'}
	fbMbTcpPortControllIn		:	fbMbTcpPortControll;
	{attribute 'VAR_IN_OUT_AS_POINTER'}
	fbMbSerialPortControllIn	:	fbMbSerialPortControll;
END_VAR
    Rectangle (0,0 160x150)
    Rectangle (0,40 160x115)
    Group (5,45 150x50)
        OnMouseClick:  Dialog=VIS_ModBusServer, Parameters={usiTcpUdpSerial: 0, fbModBusServerIn: fbModBusServerIn}, OpenModal=True, OpenCentered=True
        Button (0,0 150x50)
            OnMouseClick:  Assign=ModBus, Type=Assignment
        Image (14,4 115x30), image: CtaVisSymbols.ImagePool.Modbus_Organization_Logo
        Label (39,29 100x10), "Server overview"
    Group (5,100 150x50)
        OnMouseClick:  Dialog=VIS_MODBUS_LINE, Parameters={usiTcpSerial: 0, fbMbSerialPortControllIn: fbMbSerialPortControllIn, fbMbTcpPortControllIn: fbMbTcpPortControllIn}, OpenModal=True, OpenCentered=True
        Button (0,0 150x50)
            OnMouseClick:  Assign=ModBus, Type=Assignment
        Label (42,31 100x10), "Service Line Tcp"
        Image (14,6 115x30), image: CtaVisSymbols.ImagePool.Modbus_Organization_Logo
    Image (120,0 40x40), image: CtaVisSymbols.ImagePool.close_solo_black
        OnMouseClick:  Dialog=Current Dialog, Result=OK, NumpadKeypadSet=True
    Label (5,5 100x30), "Modbus"
END_VISUALIZATION

(* text list txtPhysikalLayer (id | default)
  0 | Default
  1 | RS232
  2 | RS422
  3 | RS423
  4 | RS485 half duplex
  5 | RS485 full duplex
  6 | DMX half duplex
   |  *)

(* text list txtParity (id | default)
  0 | Default
  1 | None
  2 | Odd
  3 | Even
  4 | Mark
  5 | Space
   |  *)

(* text list txtHandshake (id | default)
  0 | Default
  1 | None
  2 | XON XOFF
  3 | DTE RTS CTS
  4 | DCE RTS CTS
  5 | DTE DSR DTR
  6 | DCE DSR DTR
  7 | RTS Lead Time
   |  *)

(* text list txtStopBits (id | default)
  0 | Default
  1 | None
  2 | Minimum
  3 | One
  4 | OneDotFive
  5 | Two
  255 | Maximum
   |  *)
